(* Logix 5000 project; controller Machine_Maintenance_Lab2 vendor 1 type 14 code 155 rev 36.11; software revision 36.00 *)

TASK MainTask (continuous, watchdog 500 ms) : MainProgram

MODULES
   Local : vendor 1 type 14 code 155 (PointIO 0, rev 36.11)
      Discrete_IO : Embedded (PointIO 1, rev 36.11, Output RPI 20 ms)
END_MODULES

PROGRAM MainProgram   (* main routine TrafficLight *)
VAR
   Clock : FBD_TIMER := (PRE := 1000);
   ClockDone_NSGEWR : BOOL;
   ClockDone_NSREWG : BOOL;
   ClockDone_NSREWY : BOOL;
   ClockDone_NSYEWR : BOOL;
   counter : COUNTER := (PRE := 5);
   CycleCounter : COUNTER := (PRE := 5);
   delay : TIMER := (PRE := 10);
   EmerDone : BOOL;
   Emergency : BOOL;
   HighCycleTimer : COUNTER := (PRE := 700);
   i_CycleDone : ALIAS FOR o_CycleDone;
   i_GreenPB : ALIAS FOR Local:1:I.Data.0;
   i_GreenPB_ConveyorStart : ALIAS FOR i_GreenPB;
   i_GreenPBLight_Conveyor1ON : ALIAS FOR o_GreenPBLight_Conveyor1ON;
   i_NightModeButton : ALIAS FOR Local:1:I.Data.3;
   i_Pause : ALIAS FOR Pause;
   i_Piston : ALIAS FOR Local:1:O.Data.2;
   i_RedPB_StopButton : ALIAS FOR Local:1:I.Data.1;
   i_RedPBLight_Conveyor2ON : ALIAS FOR o_RedPBLight_Conveyor2ON;
   i_Turnkey : ALIAS FOR Local:1:I.Data.2;
   i_Turnkey_ItemSensor : ALIAS FOR i_Turnkey;
   ItemCounter1 : COUNTER := (PRE := 5);
   ItemCounterLeft : COUNTER := (PRE := 5);
   ItemCounterRight : COUNTER := (PRE := 6);
   LowCycleTimer : COUNTER := (PRE := 300);
   MaxState : DINT;
   myClock : FBD_TIMER;
   NewCycle : BOOL;
   NightMode : BOOL;
   o_CycleDone : BOOL;
   o_EWG : ALIAS FOR Local:1:O.Data.15;
   o_EWR : ALIAS FOR Local:1:O.Data.13;
   o_EWY : ALIAS FOR Local:1:O.Data.14;
   o_GreenPBLight : ALIAS FOR Local:1:O.Data.0;
   o_GreenPBLight_Conveyor1ON : ALIAS FOR o_GreenPBLight;
   o_NSG : ALIAS FOR Local:1:O.Data.7;
   o_NSR : ALIAS FOR Local:1:O.Data.5;
   o_NSY : ALIAS FOR Local:1:O.Data.6;
   o_Piston : ALIAS FOR i_Piston;
   o_RedPBLight : ALIAS FOR Local:1:O.Data.1;
   o_RedPBLight_Conveyor2ON : ALIAS FOR o_RedPBLight;
   OS_Out : BOOL;
   Pause : BOOL;
   preStart : DINT;
   resetBit : BOOL;
   ResetDelay : TIMER := (PRE := 500);
   s_EMER : DINT;
   s_EWRNSG : DINT;
   s_EWRNSY : DINT;
   s_Night1 : DINT;
   s_Night2 : DINT;
   s_NSREWG : DINT;
   s_NSREWY : DINT;
   Start : BOOL;
   StateCounter : FBD_COUNTER;
   StateCurrent : DINT;
   StateNext : DINT;
   StatePrev : DINT;
   ThreeSecTimer : TIMER := (PRE := 3000);
   timer : TIMER := (PRE := 5000);
   timerDoneLatch : BOOL;
   TimerHighCycle : TIMER := (PRE := 700);
   TimerLowCycle : TIMER := (PRE := 300);
   timerMem : BOOL;
   timerState : DINT;
   TurnkeyOneShot : BOOL := 1;
END_VAR

ROUTINE TrafficLight   (* structured text *)
   
   RTOR(myClock);
   
   // Set clock preset
   if(s:fs) then
   	s_NSREWG := 0;
   	s_NSREWY := 1;
   	s_EWRNSG := 2;
   	s_EWRNSY := 3;
   	s_Night1 := 4;
   	s_Night2 := 5;
   	s_EMER := 6;
   	myClock.TimerEnable := 1;
   	StateCurrent := s_NSREWG;
   end_if;
   
   //Timer allows move to next state
   if(myClock.DN) then
   	myClock.Reset := 1;
   	StateCurrent := StateNext;
   else
   	myClock.Reset := 0;
   end_if;
   
   // Pause button
   if ((not i_RedPB_StopButton)) then
   	Pause := 1;
   	Start := 0;
   end_if;
   
   // Start button
   if (i_GreenPB) then
   	Start := 1;
   	Pause := 0;
   end_if;
   
   //State logic
   //NSR - EWG
   if (StateCurrent = s_NSREWG) then
   	myClock.PRE := 3000;
   	StatePrev := StateCurrent;
   	if (i_Turnkey) then
   		StateCurrent := s_EMER;
   	elsif (i_NightModeButton) then
   		StateCurrent := s_Night1;
   	else
   		o_NSR := 1;
   		o_EWG := 1;
   
   		o_NSG := 0;
   		o_NSY := 0;
   		o_EWR := 0;
   		o_EWY := 0;
   		StateNext := s_NSREWY;
   	end_if;
   end_if;
   
   //NSR - EWY
   if (StateCurrent = s_NSREWY) then
   	myClock.PRE := 2000;
   	StatePrev := StateCurrent;
   	if (i_Turnkey) then
   		StateCurrent := s_EMER;
   	elsif (i_NightModeButton) then
   		StateCurrent := s_Night1;
   	else
   		o_NSR := 1;
   		o_EWY := 1;
   
   		o_NSG := 0;
   		o_NSY := 0;
   		o_EWR := 0;
   		o_EWG := 0;
   		StateNext := s_EWRNSG;
   	end_if;
   end_if;
   
   //EWR - NSG
   if (StateCurrent = s_EWRNSG) then
   	myClock.PRE := 3000;
   	StatePrev := StateCurrent;
   	if (i_Turnkey) then
   		StateCurrent := s_EMER;
   	elsif (i_NightModeButton) then
   		StateCurrent := s_Night1;
   	else
   		o_EWR := 1;
   		o_NSG := 1;
   
   		o_NSR := 0;
   		o_NSY := 0;
   		o_EWG := 0;
   		o_EWY := 0;
   		StateNext := s_EWRNSY;
   	end_if;
   end_if;
   
   //EWR - NSY
   if (StateCurrent = s_EWRNSY) then
   	myClock.PRE := 2000;
   	StatePrev := StateCurrent;
   	if (i_Turnkey) then
   		StateCurrent := s_EMER;
   	elsif (i_NightModeButton) then
   		StateCurrent := s_Night1;
   	else
   		o_EWR := 1;
   		o_NSY := 1;
   
   		o_NSG := 0;
   		o_NSR := 0;
   		o_EWG := 0;
   		o_EWY := 0;
   		StateNext := s_NSREWG;
   	end_if;
   end_if;
   
   //Night1
   if (StateCurrent = s_Night1) then
   	myClock.PRE := 2000;
   	StatePrev := StateCurrent;
   	if (i_Turnkey) then
   		StateCurrent := s_EMER;
   	elsif (i_NightModeButton) then
   		o_NSY := 1;
   
   		o_EWR := 0;
   		o_NSG := 0;
   		o_NSR := 0;
   		o_EWG := 0;
   		o_EWY := 0;
   		StateNext := s_Night2;
   	else
   		StateCurrent := s_NSREWG;
   	end_if;
   end_if;
   
   //Night2
   if (StateCurrent = s_Night2) then
   	myClock.PRE := 2000;
   	StatePrev := StateCurrent;
   	o_EWR := 1;
   	o_NSY := 0;
   	o_NSG := 0;
   	o_NSR := 0;
   	o_EWG := 0;
   	o_EWY := 0;
   	if (i_Turnkey) then
   		StateCurrent := s_EMER;
   	elsif (i_NightModeButton) then
   		StateNext := s_Night1;
   	else
   		StateCurrent := s_NSREWG;
   	end_if;
   end_if;
   
   //EMER
   if (StateCurrent = s_EMER) then
   	if (i_Turnkey) then
   		o_NSR := 1;
   		o_EWR := 1;
   
   		o_EWG := 0;
   		o_NSG := 0;
   		o_NSY := 0;
   		o_EWY := 0;
   	else
   		StateNext := StatePrev;
   	end_if;
   end_if;
   
   
   
END_ROUTINE
END_PROGRAM
